{attribute addProperty BoxType "EL5001-0000-1021"}
{attribute addProperty Id "StatusAT %I*Status_B030DECE1621Counter_valueAT %I*UDINT32417"}
{attribute addProperty CRC "3070484329"}
{attribute addProperty SizeInBites "48"}
{attribute addProperty SizeInBytes "6"}
TYPE SSI_Inputs_B703DF69 :
STRUCT
	{attribute addProperty Name "Status"}
	Status AT %I* : Status_B030DECE;
	{attribute addProperty Name "Counter_value"}
	Counter_value AT %I* : UDINT;
END_STRUCT
END_TYPE

(* stored: Version 1.2.0.0, ProductVersion 3.1.4024.9
   DUT SSI_Inputs_B703DF69: Id {63d0c549-188b-4b75-8414-627ba63480cb} *)
